TYPE ST_JetsonTx2 :
STRUCT
END_STRUCT
END_TYPE

(* stored: Version 1.1.0.1, ProductVersion 3.1.4022.11
   DUT ST_JetsonTx2: Id {f0e2f77a-efd1-43bd-999e-b7e3cc4bd77a} *)
